(* CODESYS project sortingPlant.export

Project tree, tasks and I/O mapping:
  Device : CODESYS Control Win V3 x64, CODESYS, version 3.5.22.30
    application Application
      libraries: Standard, 3.5.22.0 (System)
      task MainTask (cyclic, interval t#20ms, priority 1) calls SFC_PRG, Control
      global variables FIO
      program Control [FBD]
      program SFC_PRG [SFC]: Emergency_active, GoToInitalPosition_active, Reset_active, Transporting_active, Transporting_entry, EndMovingX1, End_MovingX
      Symbols
*)

// Device/Application/FIO
{attribute 'qualified_only'}
VAR_GLOBAL
	//Sensors and PBs
	AtEntry:BOOL;
	AtExit:BOOL;
 	AtLeft:BOOL;
	AtLoad:BOOL; 
	AtMiddle:BOOL;
	AtRight:BOOL;
	AtUnload:BOOL; 
	Auto:BOOL;
	EmergencyStop:BOOL;
	Manual:BOOL;
	MovingX:BOOL;
	MovingZ:BOOL;
	Reset:BOOL;
	Start:BOOL;
	Stop:BOOL;
	
	// Actuators
	EntryConveyor:BOOL:=FALSE; 
	ExitConveyor:BOOL:=FALSE; 
	ForksLeft:BOOL:=FALSE; 
	ForksRight:BOOL:=FALSE;
	Lift:BOOL:=FALSE;
	LoadConveyor:BOOL:=FALSE;
	ResetLight:BOOL:=FALSE;
	StartLight:BOOL:=FALSE;
	StopLight:BOOL:=FALSE;
	TargetPosition:WORD:=0;
	UnloadConveyor:BOOL:=0;
	
	
END_VAR

// Device/Application/SFC_PRG
PROGRAM SFC_PRG
VAR
	NextPosition: WORD := 0;
	F_TRIG_0: F_TRIG;
	F_TRIG_1: F_TRIG;
END_VAR
VAR_INPUT
	SFCinit:BOOL; 
END_VAR

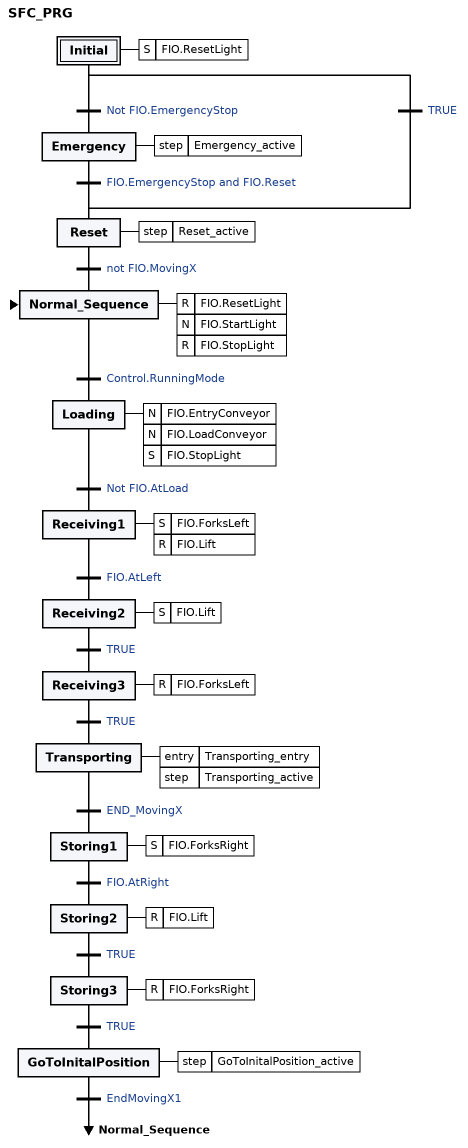
INITIAL_STEP Initial:
    FIO.ResetLight(S);
END_STEP
TRANSITION FROM Initial TO Emergency
    := Not FIO.EmergencyStop;
END_TRANSITION
STEP Emergency:
    Emergency_active(N);  // step action
END_STEP
TRANSITION FROM Emergency TO Reset
    := FIO.EmergencyStop and FIO.Reset;
END_TRANSITION
TRANSITION FROM Initial TO Reset
    := TRUE;
END_TRANSITION
STEP Reset:
    Reset_active(N);  // step action
END_STEP
TRANSITION FROM Reset TO Normal_Sequence
    := not FIO.MovingX;
END_TRANSITION
STEP Normal_Sequence:
    FIO.ResetLight(R);
    FIO.StartLight(N);
    FIO.StopLight(R);
END_STEP
TRANSITION FROM Normal_Sequence TO Loading
    := Control.RunningMode;
END_TRANSITION
STEP Loading:
    FIO.EntryConveyor(N);
    FIO.LoadConveyor(N);
    FIO.StopLight(S);
END_STEP
TRANSITION FROM Loading TO Receiving1
    := Not FIO.AtLoad;
END_TRANSITION
// macro Receiving begins
STEP Receiving1:
    FIO.ForksLeft(S);
    FIO.Lift(R);
END_STEP
TRANSITION FROM Receiving1 TO Receiving2
    := FIO.AtLeft;
END_TRANSITION
STEP Receiving2:  // min time T#2s
    FIO.Lift(S);
END_STEP
TRANSITION FROM Receiving2 TO Receiving3
    := TRUE;
END_TRANSITION
STEP Receiving3:  // min time T#2.5s
    FIO.ForksLeft(R);
END_STEP
TRANSITION FROM Receiving3 TO Transporting
    := TRUE;
END_TRANSITION
STEP Transporting:
    Transporting_entry(P1);  // entry action
    Transporting_active(N);  // step action
END_STEP
TRANSITION FROM Transporting TO Storing1
    := END_MovingX;
END_TRANSITION
// macro Storing begins
STEP Storing1:
    FIO.ForksRight(S);
END_STEP
TRANSITION FROM Storing1 TO Storing2
    := FIO.AtRight;
END_TRANSITION
STEP Storing2:  // min time T#3s
    FIO.Lift(R);
END_STEP
TRANSITION FROM Storing2 TO Storing3
    := TRUE;
END_TRANSITION
STEP Storing3:  // min time T#3s
    FIO.ForksRight(R);
END_STEP
TRANSITION FROM Storing3 TO GoToInitalPosition
    := TRUE;
END_TRANSITION
STEP GoToInitalPosition:
    GoToInitalPosition_active(N);  // step action
END_STEP
TRANSITION FROM GoToInitalPosition TO Normal_Sequence
    := EndMovingX1;
END_TRANSITION

ACTION Emergency_active:
FIO.EntryConveyor:=FALSE;
FIO.ExitConveyor:=FALSE;
FIO.ForksLeft:=FALSE;
FIO.ForksRight:=FALSE;
FIO.Lift:=FALSE;
FIO.LoadConveyor:=FALSE;
FIO.ResetLight:=FALSE;
FIO.StartLight:=FALSE;
FIO.StopLight:=FALSE;
FIO.UnloadConveyor:=FALSE; 
FIO.TargetPosition:=0;
END_ACTION

ACTION GoToInitalPosition_active:
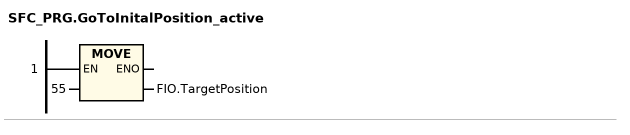
// NETWORK 1
FIO.TargetPosition := 55;
END_ACTION

ACTION Reset_active:
FIO.EntryConveyor:=FALSE;
FIO.ExitConveyor:=FALSE;
FIO.ForksLeft:=FALSE;
FIO.ForksRight:=FALSE;
FIO.Lift:=FALSE;
FIO.LoadConveyor:=FALSE;
FIO.ResetLight:=FALSE;
FIO.StartLight:=FALSE;
FIO.StopLight:=FALSE;
FIO.UnloadConveyor:=FALSE;
IF FIO.AtMiddle THEN
FIO.TargetPosition:=55;
END_IF
END_ACTION

ACTION Transporting_active:
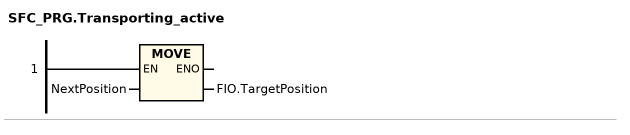
// NETWORK 1
FIO.TargetPosition := NextPosition;
END_ACTION

ACTION Transporting_entry:
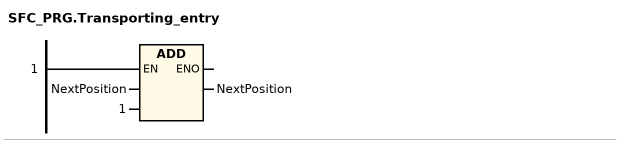
// NETWORK 1
NextPosition := NextPosition + 1;
END_ACTION

TRANSITION EndMovingX1:
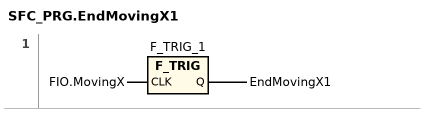
// NETWORK 1
F_TRIG_1(CLK := FIO.MovingX); // F_TRIG
EndMovingX1 := F_TRIG_1.Q;
END_TRANSITION

TRANSITION End_MovingX:
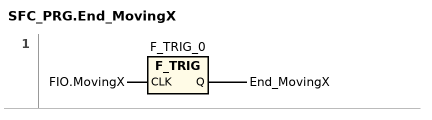
// NETWORK 1
F_TRIG_0(CLK := FIO.MovingX); // F_TRIG
End_MovingX := F_TRIG_0.Q;
END_TRANSITION

END_PROGRAM

// Device/Application/Control
PROGRAM Control
VAR
	RS_0: RS;
	RunningMode: BOOL;
	R_TRIG_0: R_TRIG;
END_VAR

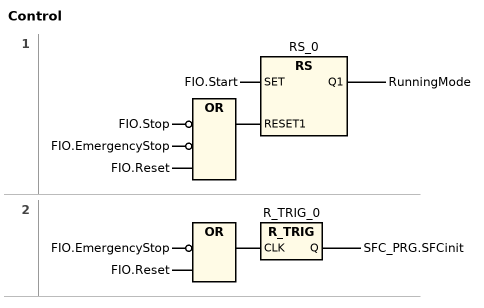
// NETWORK 1
RS_0(SET := FIO.Start, RESET1 := NOT FIO.Stop OR NOT FIO.EmergencyStop OR FIO.Reset); // RS
RunningMode := RS_0.Q1;

// NETWORK 2
R_TRIG_0(CLK := NOT FIO.EmergencyStop OR FIO.Reset); // R_TRIG
SFC_PRG.SFCinit := R_TRIG_0.Q;

END_PROGRAM
